TYPE Vec7d : ARRAY[1..7] OF LREAL; END_TYPE

(* stored: Version 1.1.0.1, ProductVersion 3.1.4024.12
   DUT Vec7d: Id {e7448c07-db7c-4e23-a784-99d23808d3ef} *)
